// Mitsubishi GX Works2 project: DemoTramCapPhoi   PLC: FX2N/FX2NC

PROGRAM MAIN
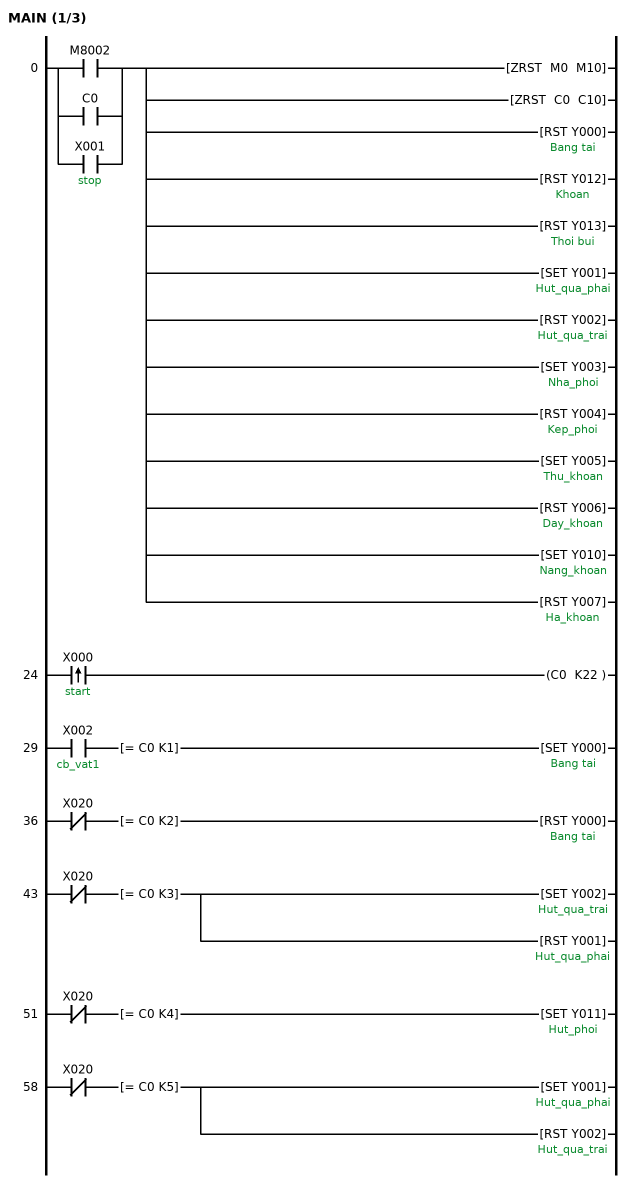
0     LD      M8002
      OR      C0
      OR      X001  ; stop
      ZRST    M0 M10
      ZRST    C0 C10
      RST     Y000  ; Bang tai
      RST     Y012  ; Khoan
      RST     Y013  ; Thoi bui
      SET     Y001  ; Hut_qua_phai
      RST     Y002  ; Hut_qua_trai
      SET     Y003  ; Nha_phoi
      RST     Y004  ; Kep_phoi
      SET     Y005  ; Thu_khoan
      RST     Y006  ; Day_khoan
      SET     Y010  ; Nang_khoan
      RST     Y007  ; Ha_khoan
24    LDP     X000  ; start
      OUT     C0 K22
29    LD      X002  ; cb_vat1
      AND=    C0 K1
      SET     Y000  ; Bang tai
36    LDI     X020
      AND=    C0 K2
      RST     Y000  ; Bang tai
43    LDI     X020
      AND=    C0 K3
      SET     Y002  ; Hut_qua_trai
      RST     Y001  ; Hut_qua_phai
51    LDI     X020
      AND=    C0 K4
      SET     Y011  ; Hut_phoi
58    LDI     X020
      AND=    C0 K5
      SET     Y001  ; Hut_qua_phai
      RST     Y002  ; Hut_qua_trai
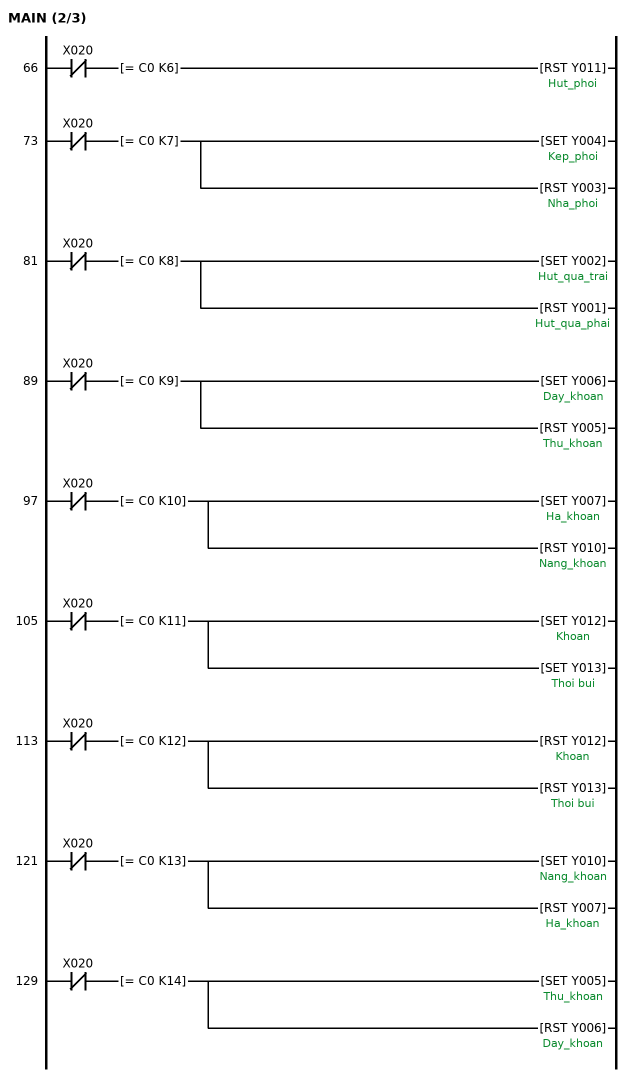
66    LDI     X020
      AND=    C0 K6
      RST     Y011  ; Hut_phoi
73    LDI     X020
      AND=    C0 K7
      SET     Y004  ; Kep_phoi
      RST     Y003  ; Nha_phoi
81    LDI     X020
      AND=    C0 K8
      SET     Y002  ; Hut_qua_trai
      RST     Y001  ; Hut_qua_phai
89    LDI     X020
      AND=    C0 K9
      SET     Y006  ; Day_khoan
      RST     Y005  ; Thu_khoan
97    LDI     X020
      AND=    C0 K10
      SET     Y007  ; Ha_khoan
      RST     Y010  ; Nang_khoan
105   LDI     X020
      AND=    C0 K11
      SET     Y012  ; Khoan
      SET     Y013  ; Thoi bui
113   LDI     X020
      AND=    C0 K12
      RST     Y012  ; Khoan
      RST     Y013  ; Thoi bui
121   LDI     X020
      AND=    C0 K13
      SET     Y010  ; Nang_khoan
      RST     Y007  ; Ha_khoan
129   LDI     X020
      AND=    C0 K14
      SET     Y005  ; Thu_khoan
      RST     Y006  ; Day_khoan
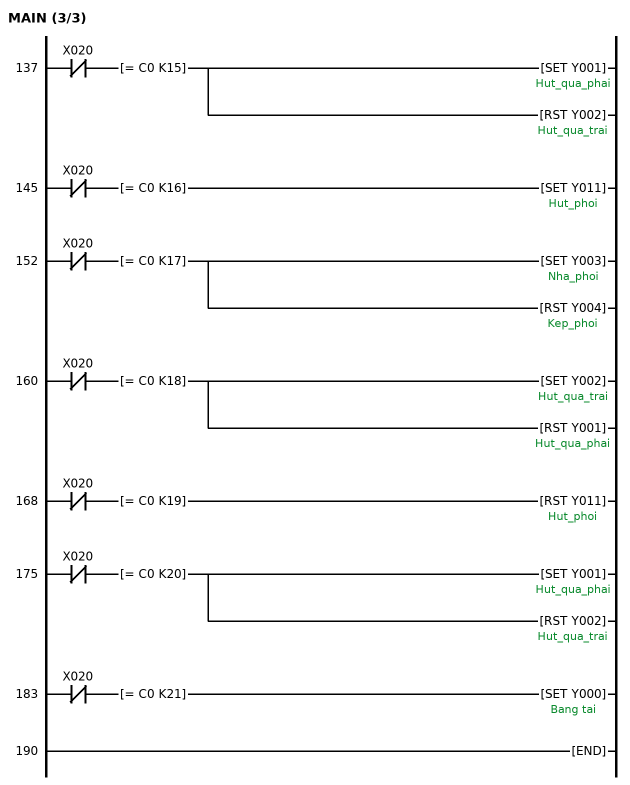
137   LDI     X020
      AND=    C0 K15
      SET     Y001  ; Hut_qua_phai
      RST     Y002  ; Hut_qua_trai
145   LDI     X020
      AND=    C0 K16
      SET     Y011  ; Hut_phoi
152   LDI     X020
      AND=    C0 K17
      SET     Y003  ; Nha_phoi
      RST     Y004  ; Kep_phoi
160   LDI     X020
      AND=    C0 K18
      SET     Y002  ; Hut_qua_trai
      RST     Y001  ; Hut_qua_phai
168   LDI     X020
      AND=    C0 K19
      RST     Y011  ; Hut_phoi
175   LDI     X020
      AND=    C0 K20
      SET     Y001  ; Hut_qua_phai
      RST     Y002  ; Hut_qua_trai
183   LDI     X020
      AND=    C0 K21
      SET     Y000  ; Bang tai
190   END
END_PROGRAM

// device comments not shown above
X003  ; cb-vat2
X004  ; cb_gap_trai
X005  ; cb_gap_phai
X007  ; cb_giu_trong
X010  ; cb_giu_ngoai
X011  ; cb_day_khoan
X012  ; cb_thu_khoan
X013  ; cb_ha_khoan
X014  ; cb_nang_khoan
